_CFC_ (* Continuous Function Chart, elements in execution order *)
#0 OR(SCHU_P2_3_UE3_VL_RESET, SCHU_P2_3_SB)
#1 SEL(UE3_VL_FILTER_ON, T#0ms, T#2s)
#2 fb_UE3_VL:ISTOK_ANALOGVH(enable: TRUE, rawValue: SCHU_P2_3_UE3_AI5, reset: #0, enableLimitCtrl: TRUE, ctrlVoltage: NOT UE3_VL_CVOLT, changeValueWithoutPower: TRUE, highRange: VL_HIGHRANGE, lowRange: VL_LOWRANGE, highLimit: SCHU_P2_3_VL_HIGHLIMIT, lowLimit: SCHU_P2_3_VL_LOWLIMIT, filterTime: #1, offset: ofset, delayEnable: VL_DELAY)
#3 SCHU_P2_3_UE3_VL_VN <= #2.presentValue
#4 SCHU_P2_3_UE3_VL_DOST <= #2.reliability
#5 SUB(SCHU_P2_3_UE3_VL_UST_OTKL, SCHU_P2_3_UE3_VL_UST_VKL)
#6 fb_SCHU_P2_3_UE3_VL_B_UST:ISTOK_GT(dost: #2.reliability, x: #2.presentValue, ust: SCHU_P2_3_UE3_VL_UST_OTKL, shkal: -, gist: #5)
#7 SCHU_P2_3_UE3_VL_B_UST <= #6.Xb
#8 SCHU_P2_3_UE3_VL_M_UST <= #6.XbN
_END_CFC_
(* the same logic as Structured Text *)
fb_UE3_VL(enable := TRUE, rawValue := SCHU_P2_3_UE3_AI5, reset := SCHU_P2_3_UE3_VL_RESET OR SCHU_P2_3_SB, enableLimitCtrl := TRUE, ctrlVoltage := NOT UE3_VL_CVOLT, changeValueWithoutPower := TRUE, highRange := VL_HIGHRANGE, lowRange := VL_LOWRANGE, highLimit := SCHU_P2_3_VL_HIGHLIMIT, lowLimit := SCHU_P2_3_VL_LOWLIMIT, filterTime := SEL(UE3_VL_FILTER_ON, T#0ms, T#2s), offset := ofset, delayEnable := VL_DELAY);
SCHU_P2_3_UE3_VL_VN := fb_UE3_VL.presentValue;
SCHU_P2_3_UE3_VL_DOST := fb_UE3_VL.reliability;
fb_SCHU_P2_3_UE3_VL_B_UST(dost := fb_UE3_VL.reliability, x := fb_UE3_VL.presentValue, ust := SCHU_P2_3_UE3_VL_UST_OTKL, gist := SCHU_P2_3_UE3_VL_UST_OTKL - SCHU_P2_3_UE3_VL_UST_VKL);
SCHU_P2_3_UE3_VL_B_UST := fb_SCHU_P2_3_UE3_VL_B_UST.Xb;
SCHU_P2_3_UE3_VL_M_UST := fb_SCHU_P2_3_UE3_VL_B_UST.XbN;
END_PROGRAM

(* POU Input/AI/YA2_POS, CFC *)
PROGRAM YA2_POS
VAR
	ofset: REAL;
	fb_YA2: ISTOK_ANALOGVH;
	Lt_otkr_zakr: ISTOK_LT;
	gt_otkr_otr: ISTOK_GT;
	fb_YA2bUST_VKL_STER_REG: ISTOK_GT;
	fb_YA2mOTKL_STER_REG: ISTOK_LT;
END_VAR
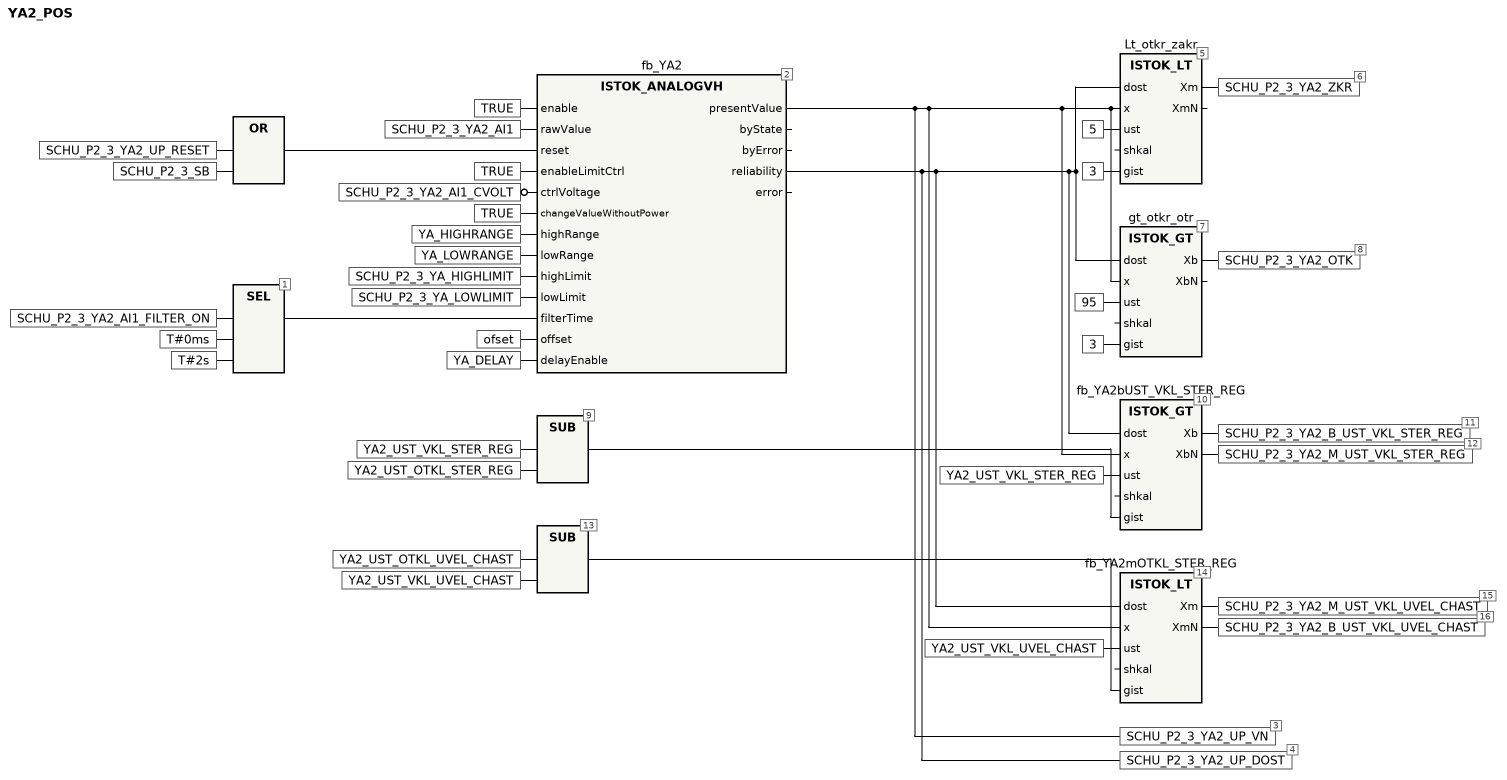
_CFC_ (* Continuous Function Chart, elements in execution order *)
#0 OR(SCHU_P2_3_YA2_UP_RESET, SCHU_P2_3_SB)
#1 SEL(SCHU_P2_3_YA2_AI1_FILTER_ON, T#0ms, T#2s)
#2 fb_YA2:ISTOK_ANALOGVH(enable: TRUE, rawValue: SCHU_P2_3_YA2_AI1, reset: #0, enableLimitCtrl: TRUE, ctrlVoltage: NOT SCHU_P2_3_YA2_AI1_CVOLT, changeValueWithoutPower: TRUE, highRange: YA_HIGHRANGE, lowRange: YA_LOWRANGE, highLimit: SCHU_P2_3_YA_HIGHLIMIT, lowLimit: SCHU_P2_3_YA_LOWLIMIT, filterTime: #1, offset: ofset, delayEnable: YA_DELAY)
#3 SCHU_P2_3_YA2_UP_VN <= #2.presentValue
#4 SCHU_P2_3_YA2_UP_DOST <= #2.reliability
#5 Lt_otkr_zakr:ISTOK_LT(dost: #2.reliability, x: #2.presentValue, ust: 5, shkal: -, gist: 3)
#6 SCHU_P2_3_YA2_ZKR <= #5.Xm
#7 gt_otkr_otr:ISTOK_GT(dost: #2.reliability, x: #2.presentValue, ust: 95, shkal: -, gist: 3)
#8 SCHU_P2_3_YA2_OTK <= #7.Xb
#9 SUB(YA2_UST_VKL_STER_REG, YA2_UST_OTKL_STER_REG)
#10 fb_YA2bUST_VKL_STER_REG:ISTOK_GT(dost: #2.reliability, x: #2.presentValue, ust: YA2_UST_VKL_STER_REG, shkal: -, gist: #9)
#11 SCHU_P2_3_YA2_B_UST_VKL_STER_REG <= #10.Xb
#12 SCHU_P2_3_YA2_M_UST_VKL_STER_REG <= #10.XbN
#13 SUB(YA2_UST_OTKL_UVEL_CHAST, YA2_UST_VKL_UVEL_CHAST)
#14 fb_YA2mOTKL_STER_REG:ISTOK_LT(dost: #2.reliability, x: #2.presentValue, ust: YA2_UST_VKL_UVEL_CHAST, shkal: -, gist: #13)
#15 SCHU_P2_3_YA2_M_UST_VKL_UVEL_CHAST <= #14.Xm
#16 SCHU_P2_3_YA2_B_UST_VKL_UVEL_CHAST <= #14.XmN
_END_CFC_
(* the same logic as Structured Text *)
fb_YA2(enable := TRUE, rawValue := SCHU_P2_3_YA2_AI1, reset := SCHU_P2_3_YA2_UP_RESET OR SCHU_P2_3_SB, enableLimitCtrl := TRUE, ctrlVoltage := NOT SCHU_P2_3_YA2_AI1_CVOLT, changeValueWithoutPower := TRUE, highRange := YA_HIGHRANGE, lowRange := YA_LOWRANGE, highLimit := SCHU_P2_3_YA_HIGHLIMIT, lowLimit := SCHU_P2_3_YA_LOWLIMIT, filterTime := SEL(SCHU_P2_3_YA2_AI1_FILTER_ON, T#0ms, T#2s), offset := ofset, delayEnable := YA_DELAY);
SCHU_P2_3_YA2_UP_VN := fb_YA2.presentValue;
SCHU_P2_3_YA2_UP_DOST := fb_YA2.reliability;
Lt_otkr_zakr(dost := fb_YA2.reliability, x := fb_YA2.presentValue, ust := 5, gist := 3);
SCHU_P2_3_YA2_ZKR := Lt_otkr_zakr.Xm;
gt_otkr_otr(dost := fb_YA2.reliability, x := fb_YA2.presentValue, ust := 95, gist := 3);
SCHU_P2_3_YA2_OTK := gt_otkr_otr.Xb;
fb_YA2bUST_VKL_STER_REG(dost := fb_YA2.reliability, x := fb_YA2.presentValue, ust := YA2_UST_VKL_STER_REG, gist := YA2_UST_VKL_STER_REG - YA2_UST_OTKL_STER_REG);
SCHU_P2_3_YA2_B_UST_VKL_STER_REG := fb_YA2bUST_VKL_STER_REG.Xb;
SCHU_P2_3_YA2_M_UST_VKL_STER_REG := fb_YA2bUST_VKL_STER_REG.XbN;
fb_YA2mOTKL_STER_REG(dost := fb_YA2.reliability, x := fb_YA2.presentValue, ust := YA2_UST_VKL_UVEL_CHAST, gist := YA2_UST_OTKL_UVEL_CHAST - YA2_UST_VKL_UVEL_CHAST);
SCHU_P2_3_YA2_M_UST_VKL_UVEL_CHAST := fb_YA2mOTKL_STER_REG.Xm;
SCHU_P2_3_YA2_B_UST_VKL_UVEL_CHAST := fb_YA2mOTKL_STER_REG.XmN;
END_PROGRAM

(* POU Input/AI/YA3_POS, CFC *)
PROGRAM YA3_POS
VAR
	fb_YA3: ISTOK_ANALOGVH;
	ofset: REAL;
	Lt_otkr_zakr: ISTOK_LT;
	gt_otkr_otr: ISTOK_GT;
	fb_YA3bUST_VKL_STER_REG: ISTOK_GT;
	fb_YA3mOTKL_STER_REG: ISTOK_LT;
END_VAR
